{attribute 'no_explicit_call' := 'Do not call the body - Stick to OOP'}
FUNCTION_BLOCK FB_XP_Feedback EXTENDS CHALET_BaseComponents.FB_CH_Feedback IMPLEMENTS I_XP_Feedback
VAR_INPUT
END_VAR
VAR_OUTPUT
END_VAR
VAR
	(* Indicates which object one would collide with. *)
	{attribute 'hide'}
	_objectInfo : ST_PlanarObjectInfoEx;
END_VAR

METHOD ClearObjectInfo : BOOL
VAR_INPUT
END_VAR
THIS^._ObjectInfo.Id := 0;
THIS^._ObjectInfo.ipObject := 0;
THIS^._ObjectInfo.ObjectType := EPlanarObjectType.None;
END_METHOD

{attribute 'monitoring':='call'}
(* Indicates which object one would collide with. *)
PROPERTY ObjectInfo : REFERENCE TO PlanarObjectInfo
GET
objectInfo REF= THIS^._objectInfo;
END_GET
SET
THIS^._objectInfo.Id			:= ObjectInfo.Id;
THIS^._objectInfo.ObjectType 	:= ObjectInfo.ObjectType;
THIS^._objectInfo.ipObject 		:= 0;
END_SET
END_PROPERTY

{attribute 'monitoring':='call'}
(* Indicates which object one would collide with. *)
PROPERTY ObjectInfoEx : REFERENCE TO ST_PlanarObjectInfoEx
GET
objectInfoEx REF= THIS^._objectInfo;
END_GET
SET
THIS^._objectInfo := ObjectInfoEx;
END_SET
END_PROPERTY

END_FUNCTION_BLOCK

(* stored: Version 1.1.0.1, ProductVersion 3.1.4024.12
   POU FB_XP_Feedback: Id {67e3d560-09f1-41ce-b857-21295b33fa36}, SpecialFunc None
   Method ClearObjectInfo: Id {30a346c8-6648-4763-b232-013ac322f0e2}
   Property ObjectInfo: Id {e8eeaec2-0fbd-4a1b-b245-08ec968594b6}
   Get Get: Id {a2d652c3-c1aa-4235-a52e-b220bd96ba5b}
   Set Set: Id {56bc4194-e62a-43f7-afc6-ab7b6ebdf06b}
   Property ObjectInfoEx: Id {9136f6c2-df29-47e0-ba76-9636df880a36}
   Get Get: Id {cdb0d62e-061e-4f1f-921e-ccf3dda7ae0d}
   Set Set: Id {11859cf4-09f8-4b5f-8585-f342b130d73a} *)
